// TIA Portal V17 export
// export: Created 2023-08-29T18:06:39.3261683Z, ExportSetting WithDefaults, DisplayName Totally Integrated Automation Portal, DisplayVersion V17 Update 5, DisplayName TIA Portal Openness, DisplayVersion V17 Update 5, DisplayName TIA Portal Teamcenter Gateway, DisplayVersion V17 Update 5, DisplayName TIA Portal Version Control Interface, DisplayVersion V17, DisplayName Simotion SCOUT TIA, DisplayVersion 5.4.3.0, DisplayName TIA Portal Test Suite Advanced, DisplayVersion V17 Update 1, DisplayName SIMOCODE ES, DisplayVersion V17 Update 5, DisplayName SINAMICS Startdrive Advanced, DisplayVersion V17 SP1, DisplayName SINAMICS Startdrive G130, G150, S120, S150, SINAMICS MV, S210, DisplayVersion V17 SP1, DisplayName SINAMICS Startdrive G110M, G120, G120C, G120D, G120P, G115D, DisplayVersion V17 SP1, DisplayName SIRIUS Safety ES, DisplayVersion V17 Update 5, DisplayName STEP 7 Professional, DisplayVersion V17 Update 5, DisplayName STEP 7 CFC, DisplayVersion V17 Update 1, DisplayName STEP 7 Safety, DisplayVersion V17, DisplayName WinCC Advanced, DisplayVersion V17 Update 5, DisplayName SIMATIC Visualization Architect, DisplayVersion V17 Update 5
FUNCTION "04_ESTOP" : Void   // FC5, F_FBD
TITLE = EMERGENCY STOP
{ S7_Optimized_Access := 'TRUE' }
VERSION : 0.1
// stored: AutoNumber true, IsIECCheckEnabled false, UDAEnableTagReadback false
BEGIN

REGION Network 1: ^S1 | Sorter COY Upper [=SC01]
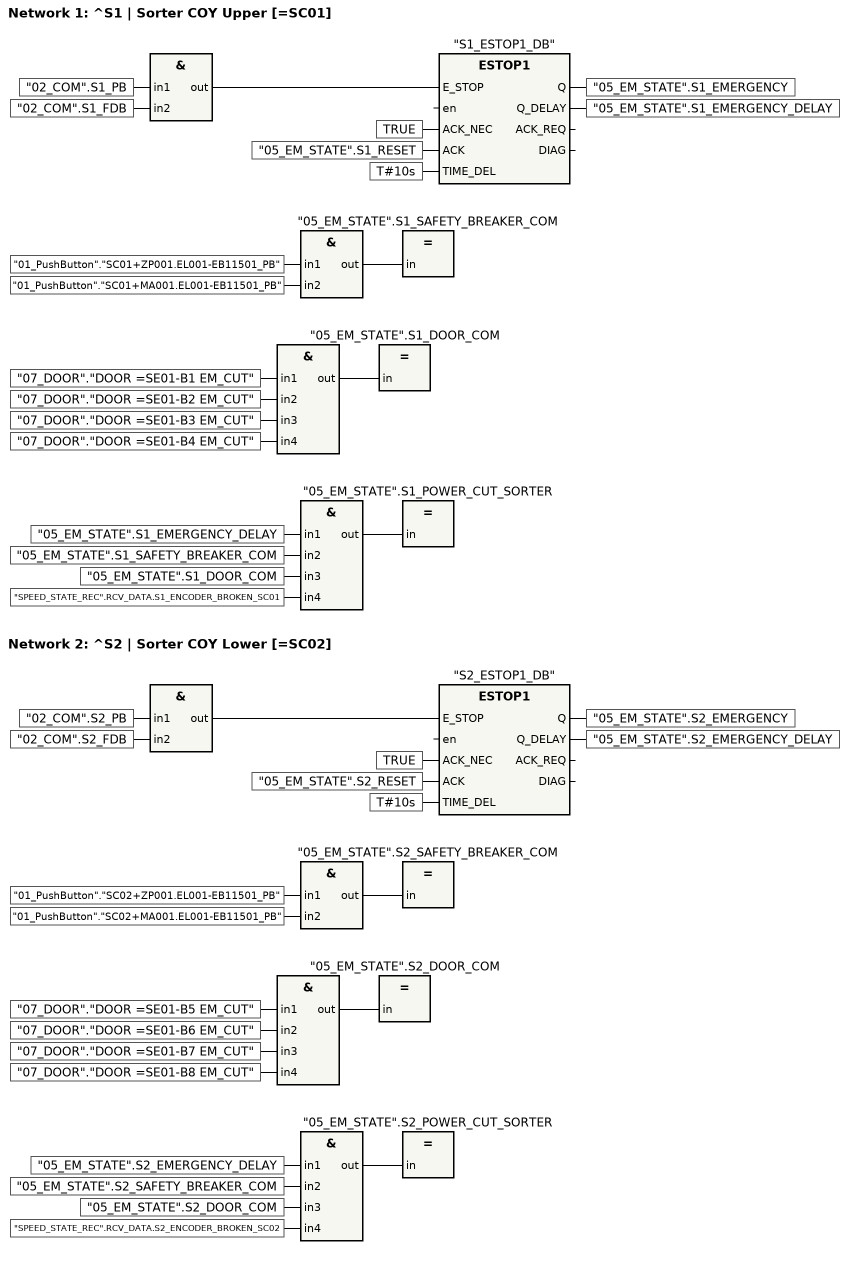
   "S1_ESTOP1_DB"(E_STOP := "02_COM".S1_PB AND "02_COM".S1_FDB,   // ESTOP1
                  ACK_NEC := TRUE,
                  ACK := "05_EM_STATE".S1_RESET,
                  TIME_DEL := T#10s,
                  Q => "05_EM_STATE".S1_EMERGENCY,
                  Q_DELAY => "05_EM_STATE".S1_EMERGENCY_DELAY);
   "05_EM_STATE".S1_SAFETY_BREAKER_COM := "01_PushButton"."SC01+ZP001.EL001-EB11501_PB" AND "01_PushButton"."SC01+MA001.EL001-EB11501_PB";
   "05_EM_STATE".S1_DOOR_COM := "07_DOOR"."DOOR =SE01-B1 EM_CUT" AND "07_DOOR"."DOOR =SE01-B2 EM_CUT" AND "07_DOOR"."DOOR =SE01-B3 EM_CUT" AND "07_DOOR"."DOOR =SE01-B4 EM_CUT";
   "05_EM_STATE".S1_POWER_CUT_SORTER := "05_EM_STATE".S1_EMERGENCY_DELAY AND "05_EM_STATE".S1_SAFETY_BREAKER_COM AND "05_EM_STATE".S1_DOOR_COM AND "SPEED_STATE_REC".RCV_DATA.S1_ENCODER_BROKEN_SC01;
END_REGION

REGION Network 2: ^S2 | Sorter COY Lower [=SC02]
   "S2_ESTOP1_DB"(E_STOP := "02_COM".S2_PB AND "02_COM".S2_FDB,   // ESTOP1
                  ACK_NEC := TRUE,
                  ACK := "05_EM_STATE".S2_RESET,
                  TIME_DEL := T#10s,
                  Q => "05_EM_STATE".S2_EMERGENCY,
                  Q_DELAY => "05_EM_STATE".S2_EMERGENCY_DELAY);
   "05_EM_STATE".S2_SAFETY_BREAKER_COM := "01_PushButton"."SC02+ZP001.EL001-EB11501_PB" AND "01_PushButton"."SC02+MA001.EL001-EB11501_PB";
   "05_EM_STATE".S2_DOOR_COM := "07_DOOR"."DOOR =SE01-B5 EM_CUT" AND "07_DOOR"."DOOR =SE01-B6 EM_CUT" AND "07_DOOR"."DOOR =SE01-B7 EM_CUT" AND "07_DOOR"."DOOR =SE01-B8 EM_CUT";
   "05_EM_STATE".S2_POWER_CUT_SORTER := "05_EM_STATE".S2_EMERGENCY_DELAY AND "05_EM_STATE".S2_SAFETY_BREAKER_COM AND "05_EM_STATE".S2_DOOR_COM AND "SPEED_STATE_REC".RCV_DATA.S2_ENCODER_BROKEN_SC02;
END_REGION

REGION Network 3: ^S3 | Sorter FLY Upper [=SF03]
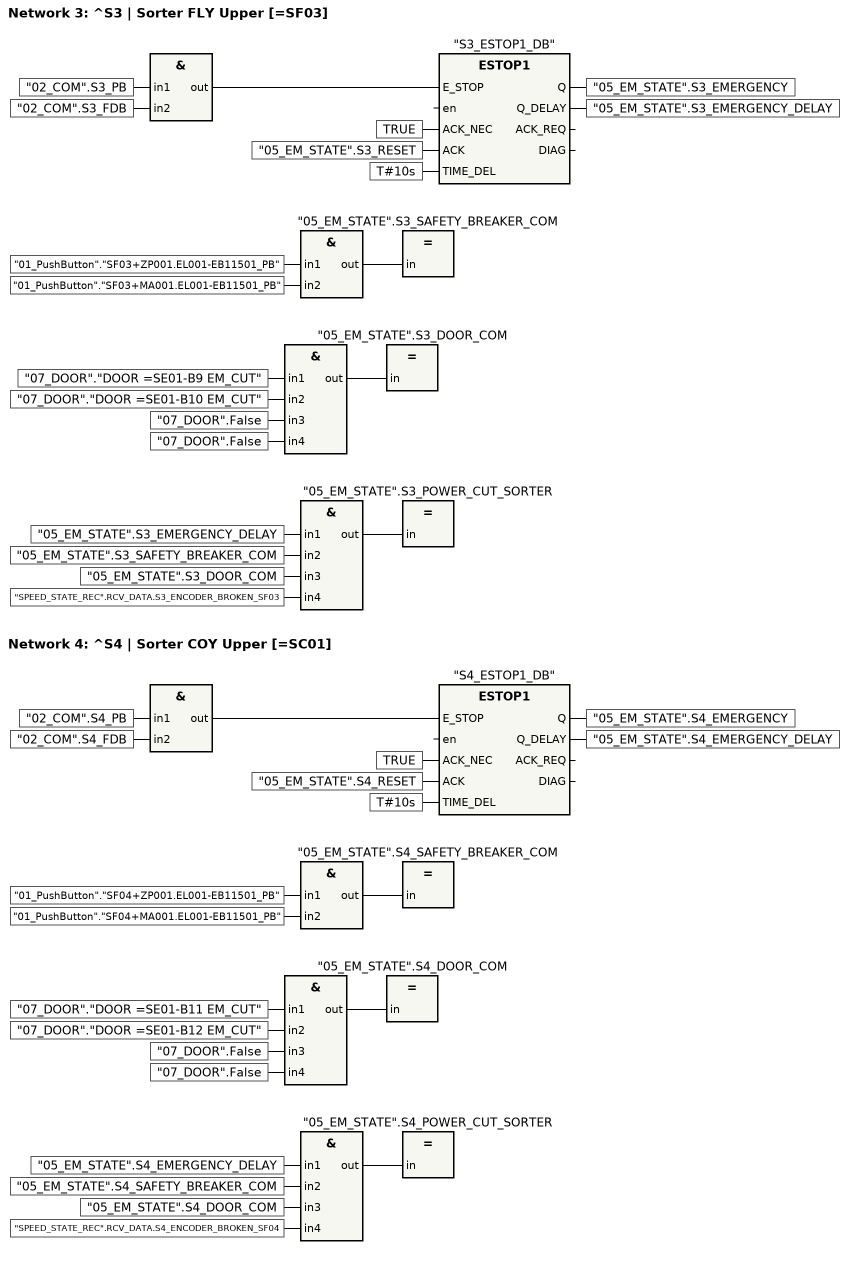
   "S3_ESTOP1_DB"(E_STOP := "02_COM".S3_PB AND "02_COM".S3_FDB,   // ESTOP1
                  ACK_NEC := TRUE,
                  ACK := "05_EM_STATE".S3_RESET,
                  TIME_DEL := T#10s,
                  Q => "05_EM_STATE".S3_EMERGENCY,
                  Q_DELAY => "05_EM_STATE".S3_EMERGENCY_DELAY);
   "05_EM_STATE".S3_SAFETY_BREAKER_COM := "01_PushButton"."SF03+ZP001.EL001-EB11501_PB" AND "01_PushButton"."SF03+MA001.EL001-EB11501_PB";
   "05_EM_STATE".S3_DOOR_COM := "07_DOOR"."DOOR =SE01-B9 EM_CUT" AND "07_DOOR"."DOOR =SE01-B10 EM_CUT" AND "07_DOOR".False AND "07_DOOR".False;
   "05_EM_STATE".S3_POWER_CUT_SORTER := "05_EM_STATE".S3_EMERGENCY_DELAY AND "05_EM_STATE".S3_SAFETY_BREAKER_COM AND "05_EM_STATE".S3_DOOR_COM AND "SPEED_STATE_REC".RCV_DATA.S3_ENCODER_BROKEN_SF03;
END_REGION

REGION Network 4: ^S4 | Sorter COY Upper [=SC01]
   "S4_ESTOP1_DB"(E_STOP := "02_COM".S4_PB AND "02_COM".S4_FDB,   // ESTOP1
                  ACK_NEC := TRUE,
                  ACK := "05_EM_STATE".S4_RESET,
                  TIME_DEL := T#10s,
                  Q => "05_EM_STATE".S4_EMERGENCY,
                  Q_DELAY => "05_EM_STATE".S4_EMERGENCY_DELAY);
   "05_EM_STATE".S4_SAFETY_BREAKER_COM := "01_PushButton"."SF04+ZP001.EL001-EB11501_PB" AND "01_PushButton"."SF04+MA001.EL001-EB11501_PB";
   "05_EM_STATE".S4_DOOR_COM := "07_DOOR"."DOOR =SE01-B11 EM_CUT" AND "07_DOOR"."DOOR =SE01-B12 EM_CUT" AND "07_DOOR".False AND "07_DOOR".False;
   "05_EM_STATE".S4_POWER_CUT_SORTER := "05_EM_STATE".S4_EMERGENCY_DELAY AND "05_EM_STATE".S4_SAFETY_BREAKER_COM AND "05_EM_STATE".S4_DOOR_COM AND "SPEED_STATE_REC".RCV_DATA.S4_ENCODER_BROKEN_SF04;
END_REGION

REGION Network 5: >A1 | AREA 1 - INTRO+UPSTREAM COY WEST
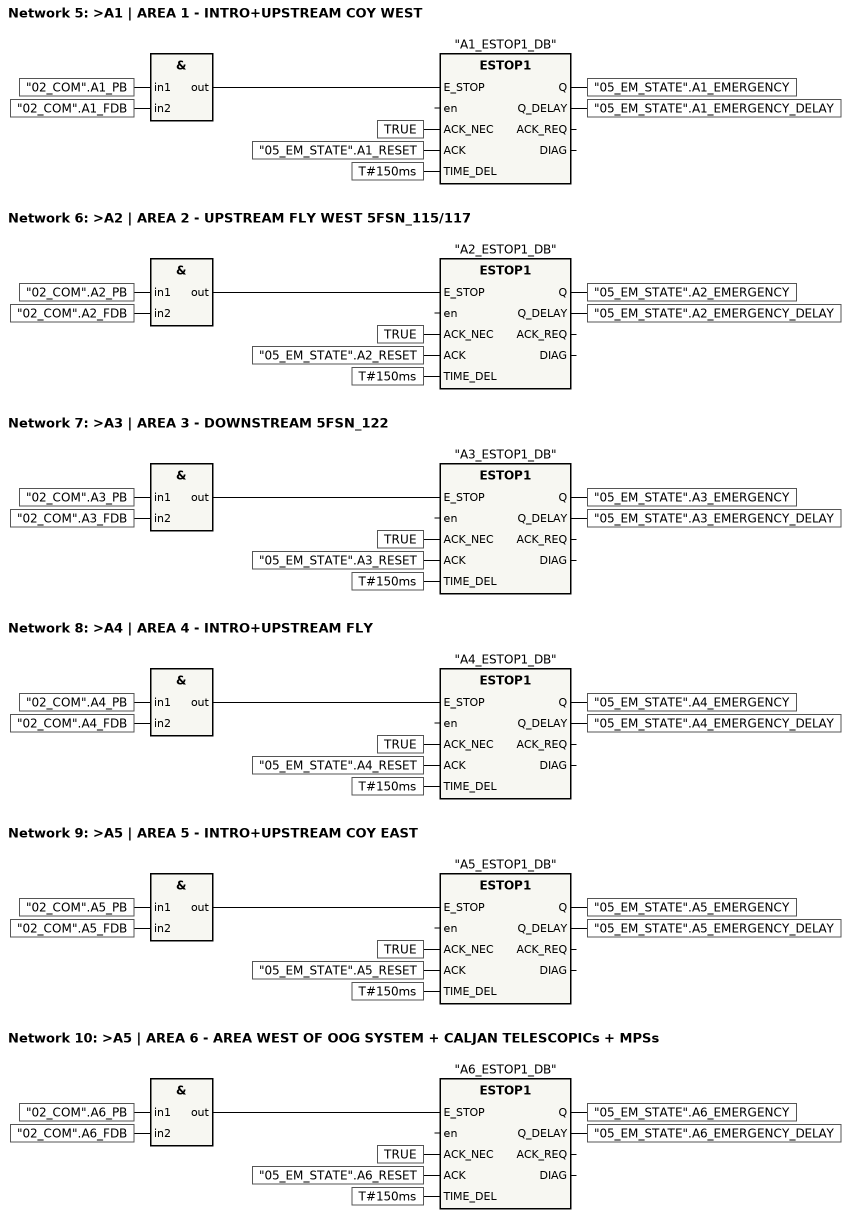
   "A1_ESTOP1_DB"(E_STOP := "02_COM".A1_PB AND "02_COM".A1_FDB,   // ESTOP1
                  ACK_NEC := TRUE,
                  ACK := "05_EM_STATE".A1_RESET,
                  TIME_DEL := T#150ms,
                  Q => "05_EM_STATE".A1_EMERGENCY,
                  Q_DELAY => "05_EM_STATE".A1_EMERGENCY_DELAY);
END_REGION

REGION Network 6: >A2 | AREA 2 - UPSTREAM FLY WEST 5FSN_115/117
   "A2_ESTOP1_DB"(E_STOP := "02_COM".A2_PB AND "02_COM".A2_FDB,   // ESTOP1
                  ACK_NEC := TRUE,
                  ACK := "05_EM_STATE".A2_RESET,
                  TIME_DEL := T#150ms,
                  Q => "05_EM_STATE".A2_EMERGENCY,
                  Q_DELAY => "05_EM_STATE".A2_EMERGENCY_DELAY);
END_REGION

REGION Network 7: >A3 | AREA 3 - DOWNSTREAM 5FSN_122
   "A3_ESTOP1_DB"(E_STOP := "02_COM".A3_PB AND "02_COM".A3_FDB,   // ESTOP1
                  ACK_NEC := TRUE,
                  ACK := "05_EM_STATE".A3_RESET,
                  TIME_DEL := T#150ms,
                  Q => "05_EM_STATE".A3_EMERGENCY,
                  Q_DELAY => "05_EM_STATE".A3_EMERGENCY_DELAY);
END_REGION

REGION Network 8: >A4 | AREA 4 - INTRO+UPSTREAM FLY
   "A4_ESTOP1_DB"(E_STOP := "02_COM".A4_PB AND "02_COM".A4_FDB,   // ESTOP1
                  ACK_NEC := TRUE,
                  ACK := "05_EM_STATE".A4_RESET,
                  TIME_DEL := T#150ms,
                  Q => "05_EM_STATE".A4_EMERGENCY,
                  Q_DELAY => "05_EM_STATE".A4_EMERGENCY_DELAY);
END_REGION

REGION Network 9: >A5 | AREA 5 - INTRO+UPSTREAM COY EAST
   "A5_ESTOP1_DB"(E_STOP := "02_COM".A5_PB AND "02_COM".A5_FDB,   // ESTOP1
                  ACK_NEC := TRUE,
                  ACK := "05_EM_STATE".A5_RESET,
                  TIME_DEL := T#150ms,
                  Q => "05_EM_STATE".A5_EMERGENCY,
                  Q_DELAY => "05_EM_STATE".A5_EMERGENCY_DELAY);
END_REGION

REGION Network 10: >A5 | AREA 6 - AREA WEST OF OOG SYSTEM + CALJAN TELESCOPICs + MPSs
   "A6_ESTOP1_DB"(E_STOP := "02_COM".A6_PB AND "02_COM".A6_FDB,   // ESTOP1
                  ACK_NEC := TRUE,
                  ACK := "05_EM_STATE".A6_RESET,
                  TIME_DEL := T#150ms,
                  Q => "05_EM_STATE".A6_EMERGENCY,
                  Q_DELAY => "05_EM_STATE".A6_EMERGENCY_DELAY);
END_REGION

REGION Network 11: >A5 | AREA 7 - AREA EAST OF OOG SYSTEM + CALJAN TELESCOPICs + MPSs
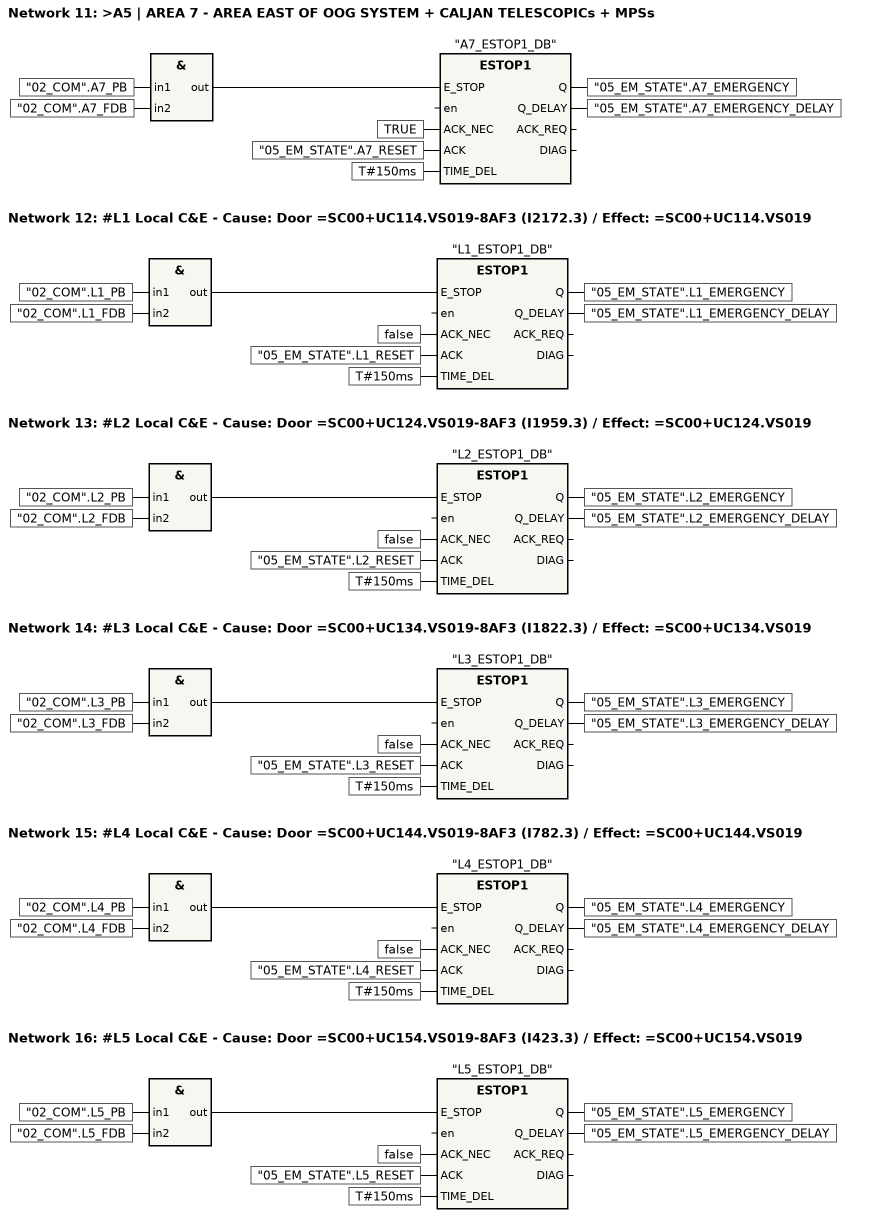
   "A7_ESTOP1_DB"(E_STOP := "02_COM".A7_PB AND "02_COM".A7_FDB,   // ESTOP1
                  ACK_NEC := TRUE,
                  ACK := "05_EM_STATE".A7_RESET,
                  TIME_DEL := T#150ms,
                  Q => "05_EM_STATE".A7_EMERGENCY,
                  Q_DELAY => "05_EM_STATE".A7_EMERGENCY_DELAY);
END_REGION

REGION Network 12: #L1 Local C&E - Cause: Door =SC00+UC114.VS019-8AF3 (I2172.3) / Effect: =SC00+UC114.VS019
   "L1_ESTOP1_DB"(E_STOP := "02_COM".L1_PB AND "02_COM".L1_FDB,   // ESTOP1
                  ACK_NEC := false,
                  ACK := "05_EM_STATE".L1_RESET,
                  TIME_DEL := T#150ms,
                  Q => "05_EM_STATE".L1_EMERGENCY,
                  Q_DELAY => "05_EM_STATE".L1_EMERGENCY_DELAY);
END_REGION

REGION Network 13: #L2 Local C&E - Cause: Door =SC00+UC124.VS019-8AF3 (I1959.3) / Effect: =SC00+UC124.VS019
   "L2_ESTOP1_DB"(E_STOP := "02_COM".L2_PB AND "02_COM".L2_FDB,   // ESTOP1
                  ACK_NEC := false,
                  ACK := "05_EM_STATE".L2_RESET,
                  TIME_DEL := T#150ms,
                  Q => "05_EM_STATE".L2_EMERGENCY,
                  Q_DELAY => "05_EM_STATE".L2_EMERGENCY_DELAY);
END_REGION

REGION Network 14: #L3 Local C&E - Cause: Door =SC00+UC134.VS019-8AF3 (I1822.3) / Effect: =SC00+UC134.VS019
   "L3_ESTOP1_DB"(E_STOP := "02_COM".L3_PB AND "02_COM".L3_FDB,   // ESTOP1
                  ACK_NEC := false,
                  ACK := "05_EM_STATE".L3_RESET,
                  TIME_DEL := T#150ms,
                  Q => "05_EM_STATE".L3_EMERGENCY,
                  Q_DELAY => "05_EM_STATE".L3_EMERGENCY_DELAY);
END_REGION

REGION Network 15: #L4 Local C&E - Cause: Door =SC00+UC144.VS019-8AF3 (I782.3) / Effect: =SC00+UC144.VS019
   "L4_ESTOP1_DB"(E_STOP := "02_COM".L4_PB AND "02_COM".L4_FDB,   // ESTOP1
                  ACK_NEC := false,
                  ACK := "05_EM_STATE".L4_RESET,
                  TIME_DEL := T#150ms,
                  Q => "05_EM_STATE".L4_EMERGENCY,
                  Q_DELAY => "05_EM_STATE".L4_EMERGENCY_DELAY);
END_REGION

REGION Network 16: #L5 Local C&E - Cause: Door =SC00+UC154.VS019-8AF3 (I423.3) / Effect: =SC00+UC154.VS019
   "L5_ESTOP1_DB"(E_STOP := "02_COM".L5_PB AND "02_COM".L5_FDB,   // ESTOP1
                  ACK_NEC := false,
                  ACK := "05_EM_STATE".L5_RESET,
                  TIME_DEL := T#150ms,
                  Q => "05_EM_STATE".L5_EMERGENCY,
                  Q_DELAY => "05_EM_STATE".L5_EMERGENCY_DELAY);
END_REGION

REGION Network 17: #L6 Local C&E - Cause: Door =SC00+UC164.VS019-8AF3 (I114.3) / Effect: =SC00+UC164.VS019
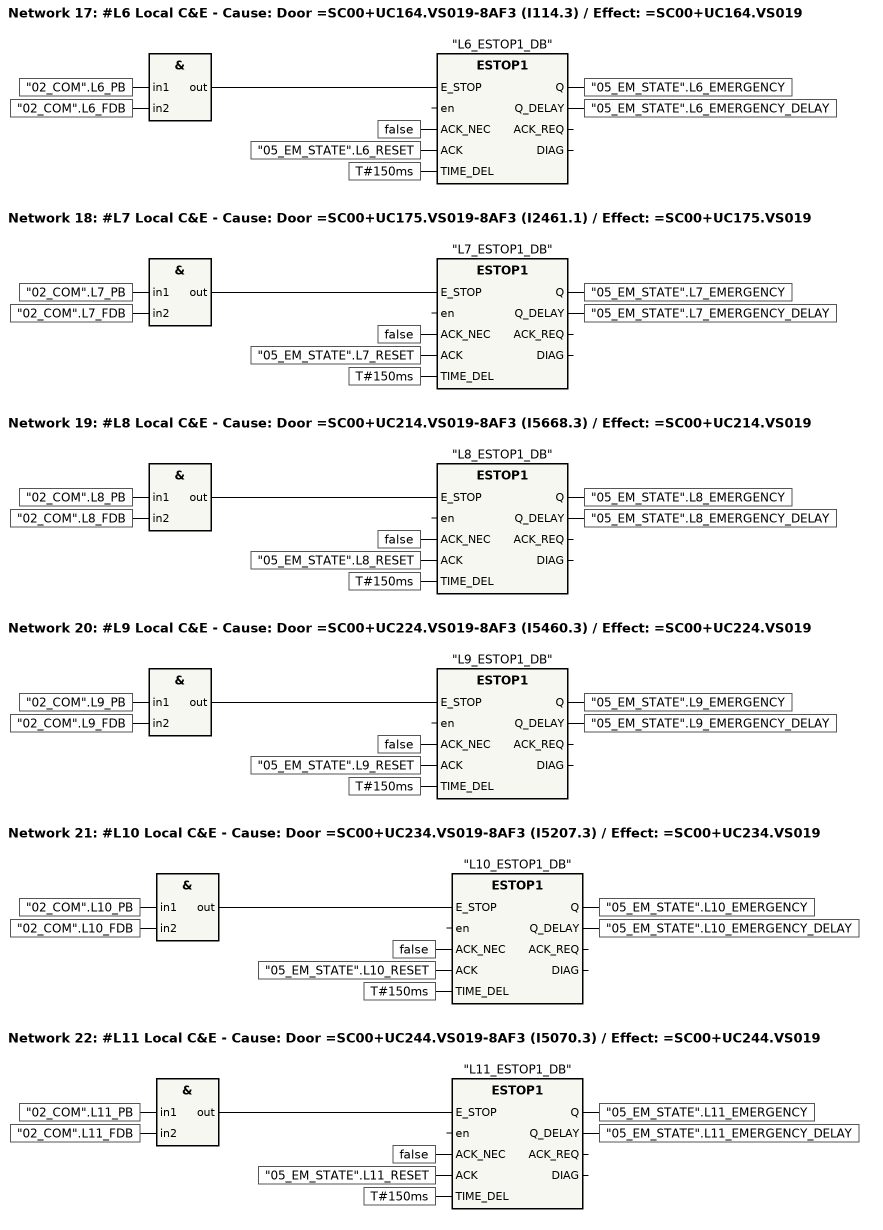
   "L6_ESTOP1_DB"(E_STOP := "02_COM".L6_PB AND "02_COM".L6_FDB,   // ESTOP1
                  ACK_NEC := false,
                  ACK := "05_EM_STATE".L6_RESET,
                  TIME_DEL := T#150ms,
                  Q => "05_EM_STATE".L6_EMERGENCY,
                  Q_DELAY => "05_EM_STATE".L6_EMERGENCY_DELAY);
END_REGION

REGION Network 18: #L7 Local C&E - Cause: Door =SC00+UC175.VS019-8AF3 (I2461.1) / Effect: =SC00+UC175.VS019
   "L7_ESTOP1_DB"(E_STOP := "02_COM".L7_PB AND "02_COM".L7_FDB,   // ESTOP1
                  ACK_NEC := false,
                  ACK := "05_EM_STATE".L7_RESET,
                  TIME_DEL := T#150ms,
                  Q => "05_EM_STATE".L7_EMERGENCY,
                  Q_DELAY => "05_EM_STATE".L7_EMERGENCY_DELAY);
END_REGION

REGION Network 19: #L8 Local C&E - Cause: Door =SC00+UC214.VS019-8AF3 (I5668.3) / Effect: =SC00+UC214.VS019
   "L8_ESTOP1_DB"(E_STOP := "02_COM".L8_PB AND "02_COM".L8_FDB,   // ESTOP1
                  ACK_NEC := false,
                  ACK := "05_EM_STATE".L8_RESET,
                  TIME_DEL := T#150ms,
                  Q => "05_EM_STATE".L8_EMERGENCY,
                  Q_DELAY => "05_EM_STATE".L8_EMERGENCY_DELAY);
END_REGION

REGION Network 20: #L9 Local C&E - Cause: Door =SC00+UC224.VS019-8AF3 (I5460.3) / Effect: =SC00+UC224.VS019
   "L9_ESTOP1_DB"(E_STOP := "02_COM".L9_PB AND "02_COM".L9_FDB,   // ESTOP1
                  ACK_NEC := false,
                  ACK := "05_EM_STATE".L9_RESET,
                  TIME_DEL := T#150ms,
                  Q => "05_EM_STATE".L9_EMERGENCY,
                  Q_DELAY => "05_EM_STATE".L9_EMERGENCY_DELAY);
END_REGION

REGION Network 21: #L10 Local C&E - Cause: Door =SC00+UC234.VS019-8AF3 (I5207.3) / Effect: =SC00+UC234.VS019
   "L10_ESTOP1_DB"(E_STOP := "02_COM".L10_PB AND "02_COM".L10_FDB,   // ESTOP1
                   ACK_NEC := false,
                   ACK := "05_EM_STATE".L10_RESET,
                   TIME_DEL := T#150ms,
                   Q => "05_EM_STATE".L10_EMERGENCY,
                   Q_DELAY => "05_EM_STATE".L10_EMERGENCY_DELAY);
END_REGION

REGION Network 22: #L11 Local C&E - Cause: Door =SC00+UC244.VS019-8AF3 (I5070.3) / Effect: =SC00+UC244.VS019
   "L11_ESTOP1_DB"(E_STOP := "02_COM".L11_PB AND "02_COM".L11_FDB,   // ESTOP1
                   ACK_NEC := false,
                   ACK := "05_EM_STATE".L11_RESET,
                   TIME_DEL := T#150ms,
                   Q => "05_EM_STATE".L11_EMERGENCY,
                   Q_DELAY => "05_EM_STATE".L11_EMERGENCY_DELAY);
END_REGION

REGION Network 23: #L12 Local C&E - Cause: Door =SC00+UC254.VS019-8AF3 (I4862.3) / Effect: =SC00+UC254.VS019
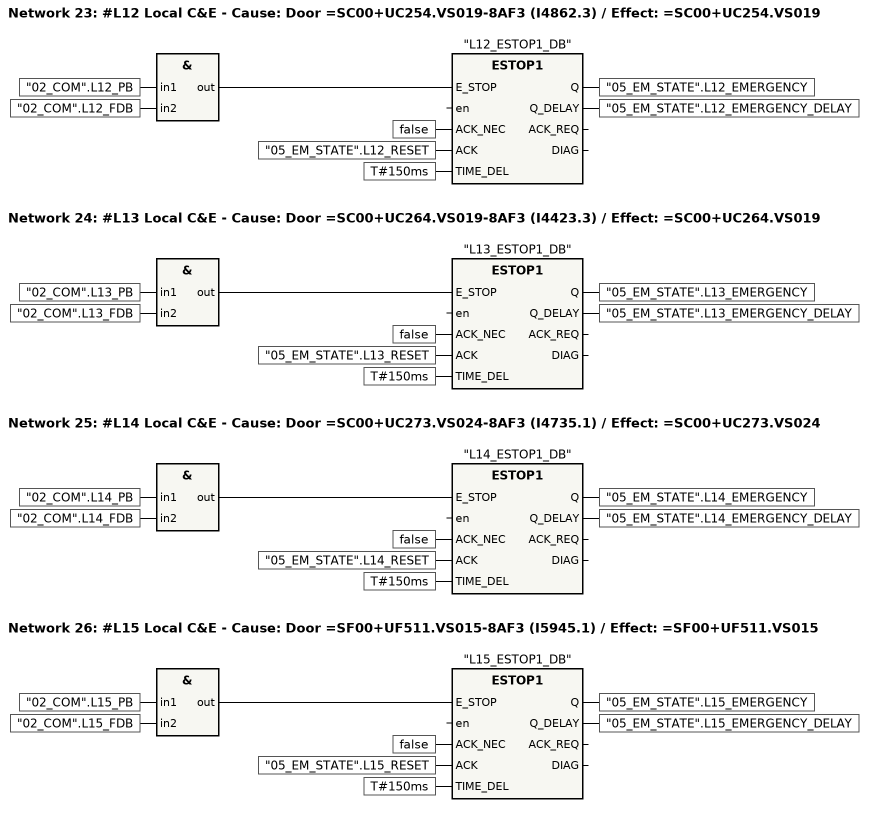
   "L12_ESTOP1_DB"(E_STOP := "02_COM".L12_PB AND "02_COM".L12_FDB,   // ESTOP1
                   ACK_NEC := false,
                   ACK := "05_EM_STATE".L12_RESET,
                   TIME_DEL := T#150ms,
                   Q => "05_EM_STATE".L12_EMERGENCY,
                   Q_DELAY => "05_EM_STATE".L12_EMERGENCY_DELAY);
END_REGION

REGION Network 24: #L13 Local C&E - Cause: Door =SC00+UC264.VS019-8AF3 (I4423.3) / Effect: =SC00+UC264.VS019
   "L13_ESTOP1_DB"(E_STOP := "02_COM".L13_PB AND "02_COM".L13_FDB,   // ESTOP1
                   ACK_NEC := false,
                   ACK := "05_EM_STATE".L13_RESET,
                   TIME_DEL := T#150ms,
                   Q => "05_EM_STATE".L13_EMERGENCY,
                   Q_DELAY => "05_EM_STATE".L13_EMERGENCY_DELAY);
END_REGION

REGION Network 25: #L14 Local C&E - Cause: Door =SC00+UC273.VS024-8AF3 (I4735.1) / Effect: =SC00+UC273.VS024
   "L14_ESTOP1_DB"(E_STOP := "02_COM".L14_PB AND "02_COM".L14_FDB,   // ESTOP1
                   ACK_NEC := false,
                   ACK := "05_EM_STATE".L14_RESET,
                   TIME_DEL := T#150ms,
                   Q => "05_EM_STATE".L14_EMERGENCY,
                   Q_DELAY => "05_EM_STATE".L14_EMERGENCY_DELAY);
END_REGION

REGION Network 26: #L15 Local C&E - Cause: Door =SF00+UF511.VS015-8AF3 (I5945.1) / Effect: =SF00+UF511.VS015
   "L15_ESTOP1_DB"(E_STOP := "02_COM".L15_PB AND "02_COM".L15_FDB,   // ESTOP1
                   ACK_NEC := false,
                   ACK := "05_EM_STATE".L15_RESET,
                   TIME_DEL := T#150ms,
                   Q => "05_EM_STATE".L15_EMERGENCY,
                   Q_DELAY => "05_EM_STATE".L15_EMERGENCY_DELAY);
END_REGION
END_FUNCTION
